// TIA Portal V19 export
ORGANIZATION_BLOCK "Main"   // OB124, LAD, ProgramCycle
TITLE = "Main Program Sweep (Cycle)"
{ S7_Optimized_Access := 'TRUE' }
// stored: SetENOAutomatically false
   VAR_INPUT
      Initial_Call : Bool;   // Initial call of this OB
      Remanence : Bool;   // =True, if remanent data are available
   END_VAR
   VAR_TEMP
      tempRHSyncBusy : Bool;
   END_VAR
BEGIN

REGION Network 1: Send Clock_Byte to subordinate system, and display Clock_Byte from subordinate system inline
   // Removed clock byte on local IO due to needing it for DQ output
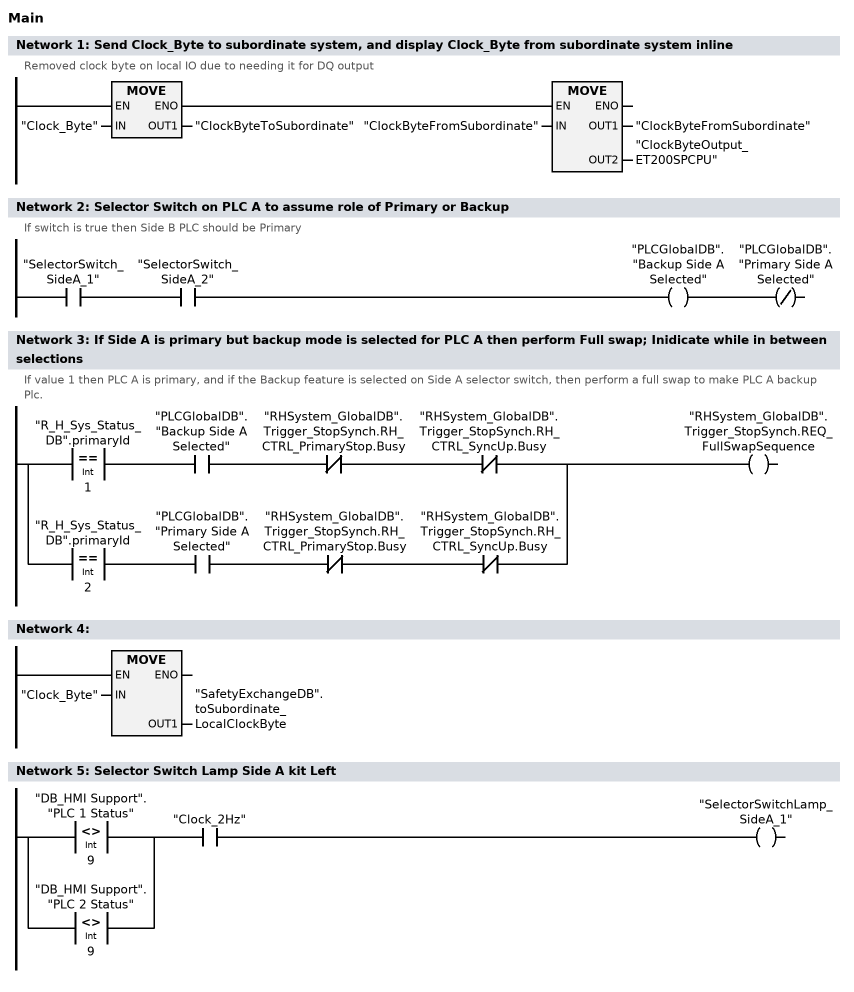
   RUNG wire#powerrail
      Move(in := "Clock_Byte", out1 => "ClockByteToSubordinate")
      Move(in := "ClockByteFromSubordinate", out1 => "ClockByteFromSubordinate", out2 => "ClockByteOutput_ET200SPCPU")
   END_RUNG
   // the same network as SCL:
   "ClockByteToSubordinate" := "Clock_Byte";
   "ClockByteFromSubordinate" := "ClockByteFromSubordinate";
   "ClockByteOutput_ET200SPCPU" := "ClockByteFromSubordinate";
END_REGION

REGION Network 2: Selector Switch on PLC A to assume role of Primary or Backup
   // If switch is true then Side B PLC should be Primary
   RUNG wire#powerrail
      Contact( "SelectorSwitch_SideA_1" )
      Contact( "SelectorSwitch_SideA_2" )
      Coil( "PLCGlobalDB"."Backup Side A Selected" )
      I_Coil( "PLCGlobalDB"."Primary Side A Selected" )
   END_RUNG
   // the same network as SCL:
   "PLCGlobalDB"."Backup Side A Selected" := "SelectorSwitch_SideA_1" AND "SelectorSwitch_SideA_2";
   "PLCGlobalDB"."Primary Side A Selected" := NOT "PLCGlobalDB"."Backup Side A Selected";
END_REGION

REGION Network 3: If Side A is primary but backup mode is selected for PLC A then perform Full swap; Inidicate while in between selections
   // If value 1 then PLC A is primary, and if the Backup feature is selected on Side A selector switch, then perform a full swap to make PLC A backup Plc.
   RUNG wire#powerrail
      { S7_Templates := "SrcType := Int" } EQ_Contact(in1 := "R_H_Sys_Status_DB".primaryId, in2 := 1)
      Contact( "PLCGlobalDB"."Backup Side A Selected" )
      I_Contact( "RHSystem_GlobalDB".Trigger_StopSynch.RH_CTRL_PrimaryStop.Busy )
      I_Contact( "RHSystem_GlobalDB".Trigger_StopSynch.RH_CTRL_SyncUp.Busy )
      wire#w1
      Coil( "RHSystem_GlobalDB".Trigger_StopSynch.REQ_FullSwapSequence )
   END_RUNG
   RUNG wire#powerrail
      { S7_Templates := "SrcType := Int" } EQ_Contact(in1 := "R_H_Sys_Status_DB".primaryId, in2 := 2)
      Contact( "PLCGlobalDB"."Primary Side A Selected" )
      I_Contact( "RHSystem_GlobalDB".Trigger_StopSynch.RH_CTRL_PrimaryStop.Busy )
      I_Contact( "RHSystem_GlobalDB".Trigger_StopSynch.RH_CTRL_SyncUp.Busy )
   END_RUNG wire#w1
   // the same network as SCL:
   "RHSystem_GlobalDB".Trigger_StopSynch.REQ_FullSwapSequence := (("R_H_Sys_Status_DB".primaryId = 1) AND "PLCGlobalDB"."Backup Side A Selected" AND NOT "RHSystem_GlobalDB".Trigger_StopSynch.RH_CTRL_PrimaryStop.Busy AND NOT "RHSystem_GlobalDB".Trigger_StopSynch.RH_CTRL_SyncUp.Busy) OR (("R_H_Sys_Status_DB".primaryId = 2) AND "PLCGlobalDB"."Primary Side A Selected" AND NOT "RHSystem_GlobalDB".Trigger_StopSynch.RH_CTRL_PrimaryStop.Busy AND NOT "RHSystem_GlobalDB".Trigger_StopSynch.RH_CTRL_SyncUp.Busy);
END_REGION

REGION Network 4
   RUNG wire#powerrail
      Move(in := "Clock_Byte", out1 => "SafetyExchangeDB".toSubordinate_LocalClockByte)
   END_RUNG
   // the same network as SCL:
   "SafetyExchangeDB".toSubordinate_LocalClockByte := "Clock_Byte";
END_REGION

REGION Network 5: Selector Switch Lamp Side A kit Left
   RUNG wire#powerrail
      { S7_Templates := "SrcType := Int" } NE_Contact(in1 := "DB_HMI Support"."PLC 1 Status", in2 := 9)
      wire#w1
      Contact( "Clock_2Hz" )
      Coil( "SelectorSwitchLamp_SideA_1" )
   END_RUNG
   RUNG wire#powerrail
      { S7_Templates := "SrcType := Int" } NE_Contact(in1 := "DB_HMI Support"."PLC 2 Status", in2 := 9)
   END_RUNG wire#w1
   // the same network as SCL:
   "SelectorSwitchLamp_SideA_1" := (("DB_HMI Support"."PLC 1 Status" <> 9) OR ("DB_HMI Support"."PLC 2 Status" <> 9)) AND "Clock_2Hz";
END_REGION
END_ORGANIZATION_BLOCK
